TYPE TankCtrl_Io_Out :
STRUCT
	bRunPump		: BOOL;
END_STRUCT
END_TYPE

(* stored: Version 1.1.0.1
   DUT TankCtrl_Io_Out: Id {5471511e-c3d1-4fb8-8289-c177f14f3234} *)
